PROGRAM MAIN
VAR
END_VAR

END_PROGRAM

(* stored: Version 1.1.0.1
   POU MAIN: Id {ed26449e-19c7-422f-814b-96d608849c0f} *)
